TYPE (* a Struct holding 2 Object IDs *)
  (* Version 1.0, 2026-05-28, franz *)
  PACKAGE isobus::UT::Q::types;
  IMPORT eclipse4diac::core::TypeHash;
  IMPORT isobus::UT::Q::const::IDs::ID_NULL;
  s2ObjectIDs : STRUCT
    u16ObjId : UINT := ID_NULL; (* Object ID Softkey *)
    u16ObjIdA : UINT := ID_NULL; (* Object ID AUX *)
  END_STRUCT;
END_TYPE
